% RSLogix 500 project I2P Project 01 - Tank 1 Process Control.RSS, saved by version 10.00.00.00 %
PROJECT "UNTITLED"    % processor: Bul.1763 MicroLogix 1100 Series B %

PROGRAM FILES
  LAD 2 "MAIN"  21 rungs  % Process Tank 1 Controls %
  LAD 3 "SIM"  18 rungs  % Simulation %

DATA FILES
  O0 OUTPUT  4 elements
  I1 INPUT  6 elements
  S2 STATUS  66 elements
  B3 BINARY  11 elements
  T4 TIMER  16 elements
  C5 COUNTER  1 elements
  R6 CONTROL  1 elements
  N7 INTEGER  1 elements
  F8 FLOAT  2 elements

LADDER 2 "MAIN"    % Process Tank 1 Controls %
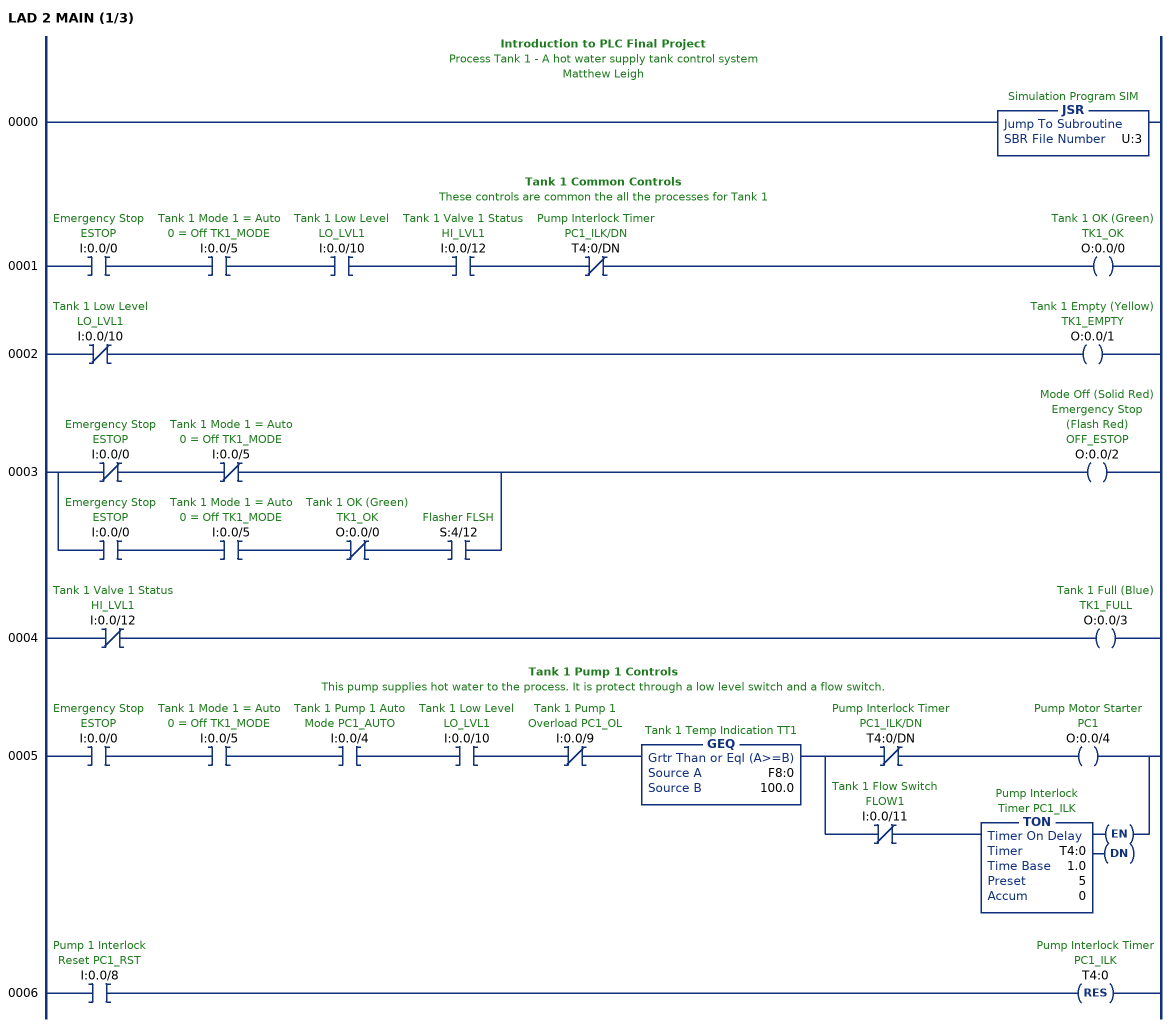
% Rung: 0 %
% TITLE: Introduction to PLC Final Project %
% Process Tank 1 - A hot water supply tank control system
% Matthew Leigh %
SOR JSR U:3 EOR
%   U:3  SIM  "Simulation Program" %
% Rung: 1 %
% TITLE: Tank 1 Common Controls %
% These controls are common the all the processes for Tank 1 %
SOR XIC I:0.0/0 XIC I:0.0/5 XIC I:0.0/10 XIC I:0.0/12 XIO T4:0/DN OTE O:0.0/0 EOR
%   I:0.0/0  ESTOP  "Emergency Stop" %
%   I:0.0/5  TK1_MODE  "Tank 1 Mode 1 = Auto 0 = Off" %
%   I:0.0/10  LO_LVL1  "Tank 1 Low Level" %
%   I:0.0/12  HI_LVL1  "Tank 1 Valve 1 Status" %
%   T4:0  PC1_ILK  "Pump Interlock Timer" %
%   O:0.0/0  TK1_OK  "Tank 1 OK (Green)" %
% Rung: 2 %
SOR XIO I:0.0/10 OTE O:0.0/1 EOR
%   I:0.0/10  LO_LVL1  "Tank 1 Low Level" %
%   O:0.0/1  TK1_EMPTY  "Tank 1 Empty (Yellow)" %
% Rung: 3 %
SOR BST XIO I:0.0/0 XIO I:0.0/5 NXB XIC I:0.0/0 XIC I:0.0/5 XIO O:0.0/0 XIC S:4/12 BND OTE O:0.0/2 EOR
%   I:0.0/0  ESTOP  "Emergency Stop" %
%   I:0.0/5  TK1_MODE  "Tank 1 Mode 1 = Auto 0 = Off" %
%   O:0.0/0  TK1_OK  "Tank 1 OK (Green)" %
%   S:4/12  FLSH  "Flasher" %
%   O:0.0/2  OFF_ESTOP  "Mode Off (Solid Red) Emergency Stop (Flash Red)" %
% Rung: 4 %
SOR XIO I:0.0/12 OTE O:0.0/3 EOR
%   I:0.0/12  HI_LVL1  "Tank 1 Valve 1 Status" %
%   O:0.0/3  TK1_FULL  "Tank 1 Full (Blue)" %
% Rung: 5 %
% TITLE: Tank 1 Pump 1 Controls %
% This pump supplies hot water to the process. It is protect through a low level switch and a flow switch. %
SOR XIC I:0.0/0 XIC I:0.0/5 XIC I:0.0/4 XIC I:0.0/10 XIO I:0.0/9 GEQ F8:0 100.0 BST XIO T4:0/DN OTE O:0.0/4 NXB XIO I:0.0/11 TON T4:0 1.0 5 0 BND EOR
%   I:0.0/0  ESTOP  "Emergency Stop" %
%   I:0.0/5  TK1_MODE  "Tank 1 Mode 1 = Auto 0 = Off" %
%   I:0.0/4  PC1_AUTO  "Tank 1 Pump 1 Auto Mode" %
%   I:0.0/10  LO_LVL1  "Tank 1 Low Level" %
%   I:0.0/9  PC1_OL  "Tank 1 Pump 1 Overload" %
%   F8:0  TT1  "Tank 1 Temp Indication" %
%   T4:0  PC1_ILK  "Pump Interlock Timer" %
%   O:0.0/4  PC1  "Pump Motor Starter" %
%   I:0.0/11  FLOW1  "Tank 1 Flow Switch" %
% Rung: 6 %
SOR XIC I:0.0/8 RES T4:0 EOR
%   I:0.0/8  PC1_RST  "Pump 1 Interlock Reset" %
%   T4:0  PC1_ILK  "Pump Interlock Timer" %

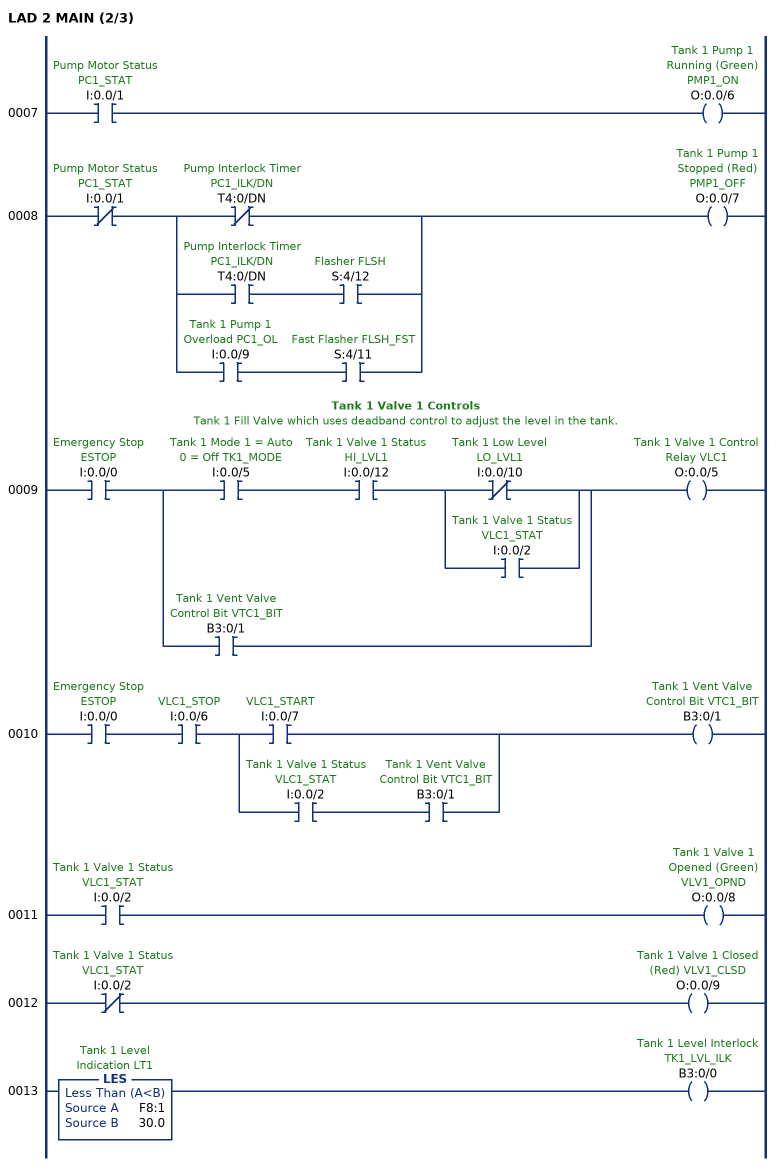
% Rung: 7 %
SOR XIC I:0.0/1 OTE O:0.0/6 EOR
%   I:0.0/1  PC1_STAT  "Pump Motor Status" %
%   O:0.0/6  PMP1_ON  "Tank 1 Pump 1 Running (Green)" %
% Rung: 8 %
SOR XIO I:0.0/1 BST XIO T4:0/DN NXB XIC T4:0/DN XIC S:4/12 NXB XIC I:0.0/9 XIC S:4/11 BND OTE O:0.0/7 EOR
%   I:0.0/1  PC1_STAT  "Pump Motor Status" %
%   T4:0  PC1_ILK  "Pump Interlock Timer" %
%   S:4/12  FLSH  "Flasher" %
%   I:0.0/9  PC1_OL  "Tank 1 Pump 1 Overload" %
%   S:4/11  FLSH_FST  "Fast Flasher" %
%   O:0.0/7  PMP1_OFF  "Tank 1 Pump 1 Stopped (Red)" %
% Rung: 9 %
% TITLE: Tank 1 Valve 1 Controls %
% Tank 1 Fill Valve which uses deadband control to adjust the level in the tank. %
SOR XIC I:0.0/0 BST XIC I:0.0/5 XIC I:0.0/12 BST XIO I:0.0/10 NXB XIC I:0.0/2 BND NXB XIC B3:0/1 BND OTE O:0.0/5 EOR
%   I:0.0/0  ESTOP  "Emergency Stop" %
%   I:0.0/5  TK1_MODE  "Tank 1 Mode 1 = Auto 0 = Off" %
%   I:0.0/12  HI_LVL1  "Tank 1 Valve 1 Status" %
%   I:0.0/10  LO_LVL1  "Tank 1 Low Level" %
%   I:0.0/2  VLC1_STAT  "Tank 1 Valve 1 Status" %
%   B3:0/1  VTC1_BIT  "Tank 1 Vent Valve Control Bit" %
%   O:0.0/5  VLC1  "Tank 1 Valve 1 Control Relay" %
% Rung: 10 %
SOR XIC I:0.0/0 XIC I:0.0/6 BST XIC I:0.0/7 NXB XIC I:0.0/2 XIC B3:0/1 BND OTE B3:0/1 EOR
%   I:0.0/0  ESTOP  "Emergency Stop" %
%   I:0.0/6  VLC1_STOP %
%   I:0.0/7  VLC1_START %
%   I:0.0/2  VLC1_STAT  "Tank 1 Valve 1 Status" %
%   B3:0/1  VTC1_BIT  "Tank 1 Vent Valve Control Bit" %
% Rung: 11 %
SOR XIC I:0.0/2 OTE O:0.0/8 EOR
%   I:0.0/2  VLC1_STAT  "Tank 1 Valve 1 Status" %
%   O:0.0/8  VLV1_OPND  "Tank 1 Valve 1 Opened (Green)" %
% Rung: 12 %
SOR XIO I:0.0/2 OTE O:0.0/9 EOR
%   I:0.0/2  VLC1_STAT  "Tank 1 Valve 1 Status" %
%   O:0.0/9  VLV1_CLSD  "Tank 1 Valve 1 Closed (Red)" %
% Rung: 13 %
SOR LES F8:1 30.0 OTE B3:0/0 EOR
%   F8:1  LT1  "Tank 1 Level Indication" %
%   B3:0/0  TK1_LVL_ILK  "Tank 1 Level Interlock" %

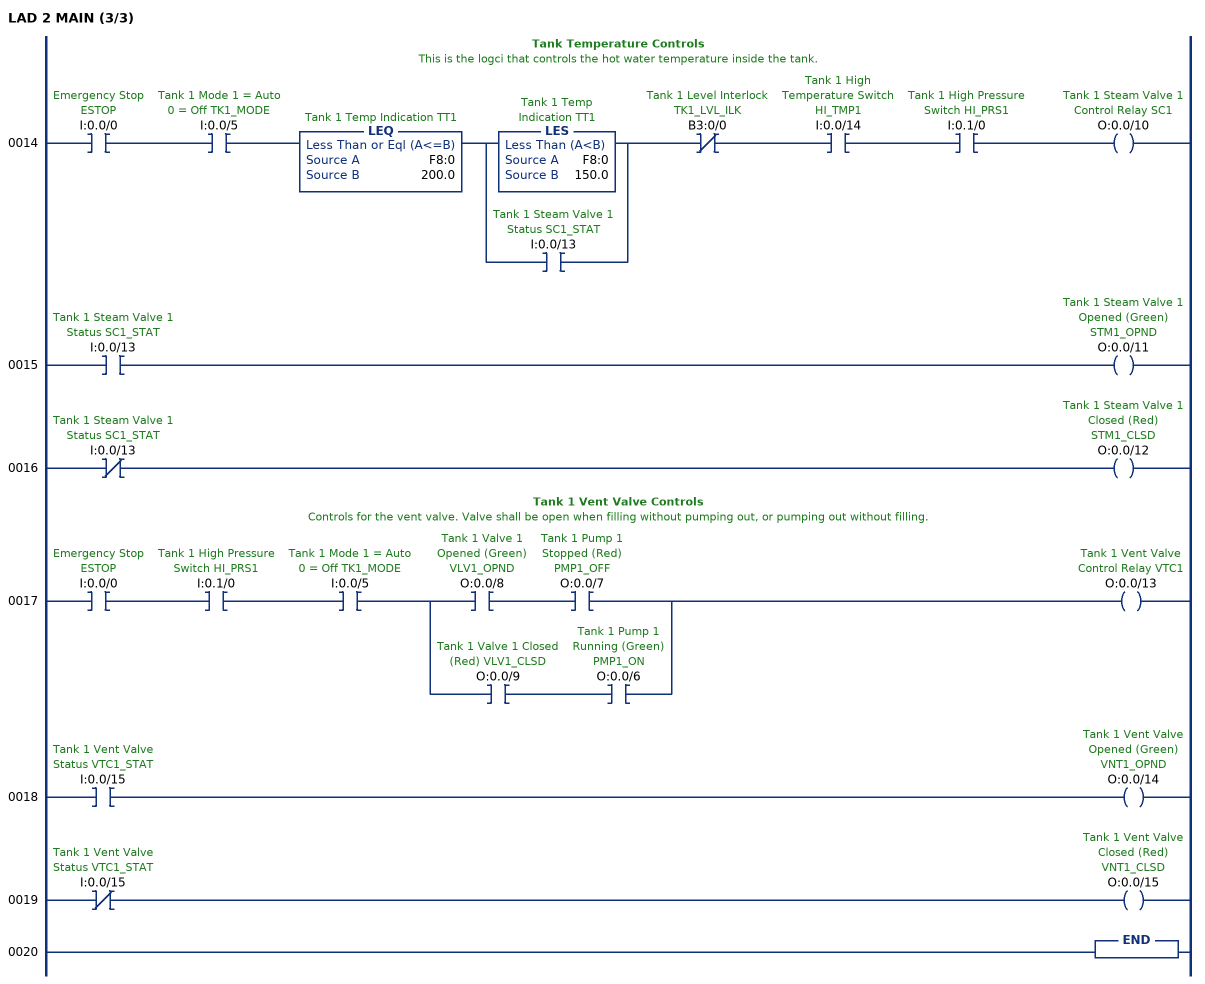
% Rung: 14 %
% TITLE: Tank Temperature Controls %
% This is the logci that controls the hot water temperature inside the tank. %
SOR XIC I:0.0/0 XIC I:0.0/5 LEQ F8:0 200.0 BST LES F8:0 150.0 NXB XIC I:0.0/13 BND XIO B3:0/0 XIC I:0.0/14 XIC I:0.1/0 OTE O:0.0/10 EOR
%   I:0.0/0  ESTOP  "Emergency Stop" %
%   I:0.0/5  TK1_MODE  "Tank 1 Mode 1 = Auto 0 = Off" %
%   F8:0  TT1  "Tank 1 Temp Indication" %
%   I:0.0/13  SC1_STAT  "Tank 1 Steam Valve 1 Status" %
%   B3:0/0  TK1_LVL_ILK  "Tank 1 Level Interlock" %
%   I:0.0/14  HI_TMP1  "Tank 1 High Temperature Switch" %
%   I:0.1/0  HI_PRS1  "Tank 1 High Pressure Switch" %
%   O:0.0/10  SC1  "Tank 1 Steam Valve 1 Control Relay" %
% Rung: 15 %
SOR XIC I:0.0/13 OTE O:0.0/11 EOR
%   I:0.0/13  SC1_STAT  "Tank 1 Steam Valve 1 Status" %
%   O:0.0/11  STM1_OPND  "Tank 1 Steam Valve 1 Opened (Green)" %
% Rung: 16 %
SOR XIO I:0.0/13 OTE O:0.0/12 EOR
%   I:0.0/13  SC1_STAT  "Tank 1 Steam Valve 1 Status" %
%   O:0.0/12  STM1_CLSD  "Tank 1 Steam Valve 1 Closed (Red)" %
% Rung: 17 %
% TITLE: Tank 1 Vent Valve Controls %
% Controls for the vent valve. Valve shall be open when filling without pumping out, or pumping out without filling. %
SOR XIC I:0.0/0 XIC I:0.1/0 XIC I:0.0/5 BST XIC O:0.0/8 XIC O:0.0/7 NXB XIC O:0.0/9 XIC O:0.0/6 BND OTE O:0.0/13 EOR
%   I:0.0/0  ESTOP  "Emergency Stop" %
%   I:0.1/0  HI_PRS1  "Tank 1 High Pressure Switch" %
%   I:0.0/5  TK1_MODE  "Tank 1 Mode 1 = Auto 0 = Off" %
%   O:0.0/8  VLV1_OPND  "Tank 1 Valve 1 Opened (Green)" %
%   O:0.0/7  PMP1_OFF  "Tank 1 Pump 1 Stopped (Red)" %
%   O:0.0/9  VLV1_CLSD  "Tank 1 Valve 1 Closed (Red)" %
%   O:0.0/6  PMP1_ON  "Tank 1 Pump 1 Running (Green)" %
%   O:0.0/13  VTC1  "Tank 1 Vent Valve Control Relay" %
% Rung: 18 %
SOR XIC I:0.0/15 OTE O:0.0/14 EOR
%   I:0.0/15  VTC1_STAT  "Tank 1 Vent Valve Status" %
%   O:0.0/14  VNT1_OPND  "Tank 1 Vent Valve Opened (Green)" %
% Rung: 19 %
SOR XIO I:0.0/15 OTE O:0.0/15 EOR
%   I:0.0/15  VTC1_STAT  "Tank 1 Vent Valve Status" %
%   O:0.0/15  VNT1_CLSD  "Tank 1 Vent Valve Closed (Red)" %
% Rung: 20 %
SOR END EOR

LADDER 3 "SIM"    % Simulation %
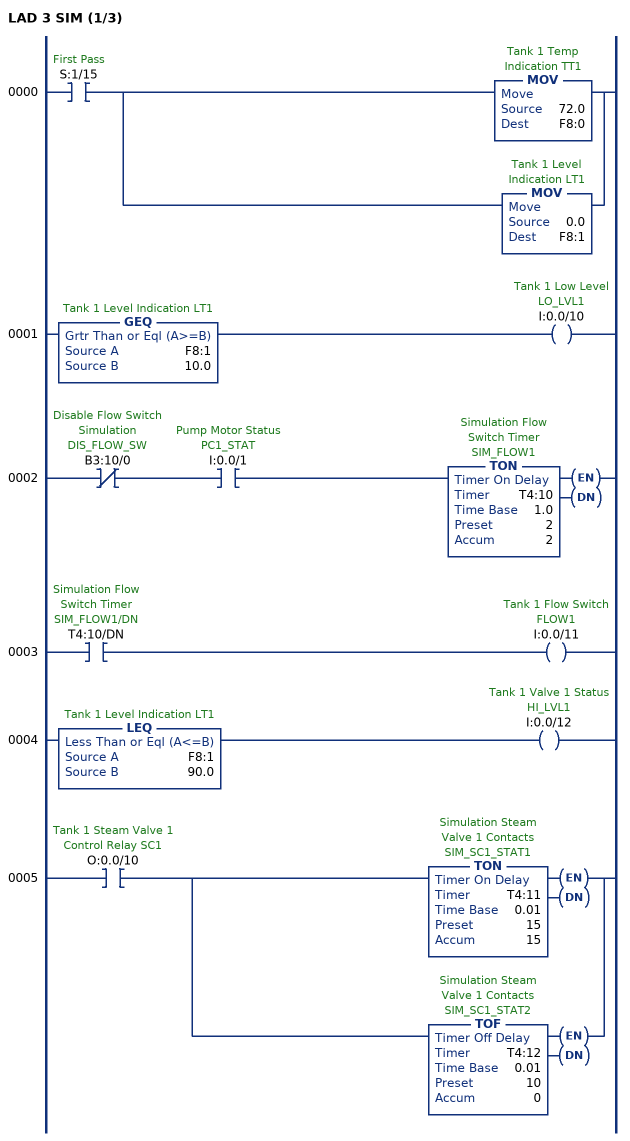
% Rung: 0 %
SOR XIC S:1/15 BST MOV 72.0 F8:0 NXB MOV 0.0 F8:1 BND EOR
%   S:1/15  "First Pass" %
%   F8:0  TT1  "Tank 1 Temp Indication" %
%   F8:1  LT1  "Tank 1 Level Indication" %
% Rung: 1 %
SOR GEQ F8:1 10.0 OTE I:0.0/10 EOR
%   F8:1  LT1  "Tank 1 Level Indication" %
%   I:0.0/10  LO_LVL1  "Tank 1 Low Level" %
% Rung: 2 %
SOR XIO B3:10/0 XIC I:0.0/1 TON T4:10 1.0 2 2 EOR
%   B3:10/0  DIS_FLOW_SW  "Disable Flow Switch Simulation" %
%   I:0.0/1  PC1_STAT  "Pump Motor Status" %
%   T4:10  SIM_FLOW1  "Simulation Flow Switch Timer" %
% Rung: 3 %
SOR XIC T4:10/DN OTE I:0.0/11 EOR
%   T4:10  SIM_FLOW1  "Simulation Flow Switch Timer" %
%   I:0.0/11  FLOW1  "Tank 1 Flow Switch" %
% Rung: 4 %
SOR LEQ F8:1 90.0 OTE I:0.0/12 EOR
%   F8:1  LT1  "Tank 1 Level Indication" %
%   I:0.0/12  HI_LVL1  "Tank 1 Valve 1 Status" %
% Rung: 5 %
SOR XIC O:0.0/10 BST TON T4:11 0.01 15 15 NXB TOF T4:12 0.01 10 0 BND EOR
%   O:0.0/10  SC1  "Tank 1 Steam Valve 1 Control Relay" %
%   T4:11  SIM_SC1_STAT1  "Simulation Steam Valve 1 Contacts" %
%   T4:12  SIM_SC1_STAT2  "Simulation Steam Valve 1 Contacts" %

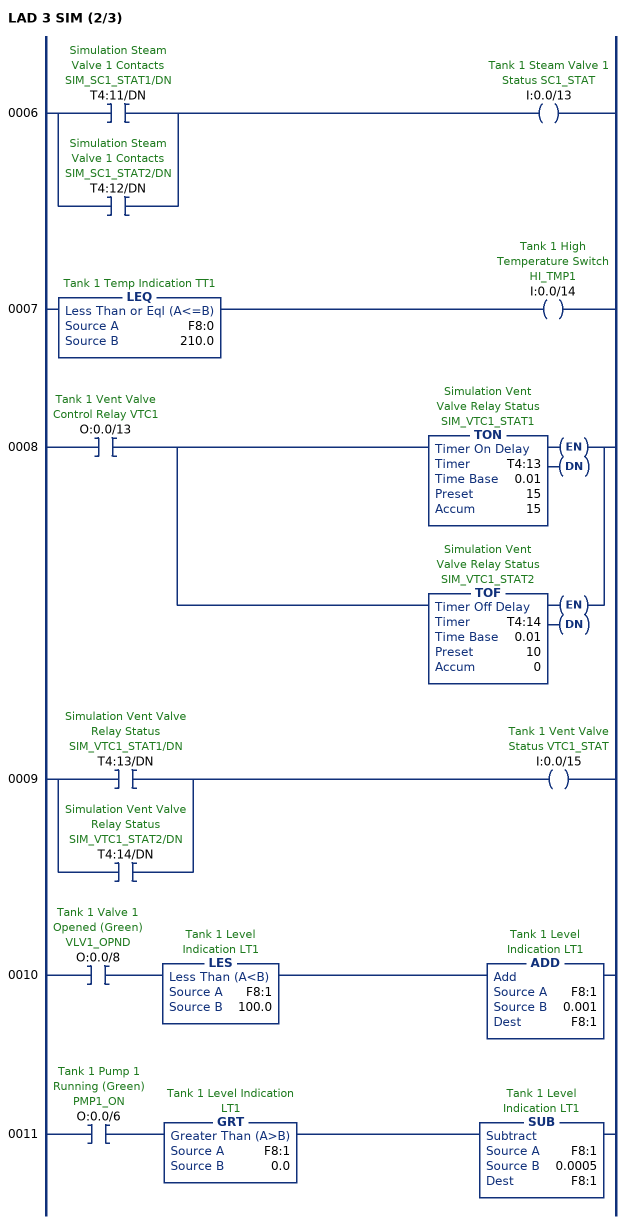
% Rung: 6 %
SOR BST XIC T4:11/DN NXB XIC T4:12/DN BND OTE I:0.0/13 EOR
%   T4:11  SIM_SC1_STAT1  "Simulation Steam Valve 1 Contacts" %
%   T4:12  SIM_SC1_STAT2  "Simulation Steam Valve 1 Contacts" %
%   I:0.0/13  SC1_STAT  "Tank 1 Steam Valve 1 Status" %
% Rung: 7 %
SOR LEQ F8:0 210.0 OTE I:0.0/14 EOR
%   F8:0  TT1  "Tank 1 Temp Indication" %
%   I:0.0/14  HI_TMP1  "Tank 1 High Temperature Switch" %
% Rung: 8 %
SOR XIC O:0.0/13 BST TON T4:13 0.01 15 15 NXB TOF T4:14 0.01 10 0 BND EOR
%   O:0.0/13  VTC1  "Tank 1 Vent Valve Control Relay" %
%   T4:13  SIM_VTC1_STAT1  "Simulation Vent Valve Relay Status" %
%   T4:14  SIM_VTC1_STAT2  "Simulation Vent Valve Relay Status" %
% Rung: 9 %
SOR BST XIC T4:13/DN NXB XIC T4:14/DN BND OTE I:0.0/15 EOR
%   T4:13  SIM_VTC1_STAT1  "Simulation Vent Valve Relay Status" %
%   T4:14  SIM_VTC1_STAT2  "Simulation Vent Valve Relay Status" %
%   I:0.0/15  VTC1_STAT  "Tank 1 Vent Valve Status" %
% Rung: 10 %
SOR XIC O:0.0/8 LES F8:1 100.0 ADD F8:1 0.001 F8:1 EOR
%   O:0.0/8  VLV1_OPND  "Tank 1 Valve 1 Opened (Green)" %
%   F8:1  LT1  "Tank 1 Level Indication" %
% Rung: 11 %
SOR XIC O:0.0/6 GRT F8:1 0.0 SUB F8:1 0.0005 F8:1 EOR
%   O:0.0/6  PMP1_ON  "Tank 1 Pump 1 Running (Green)" %
%   F8:1  LT1  "Tank 1 Level Indication" %

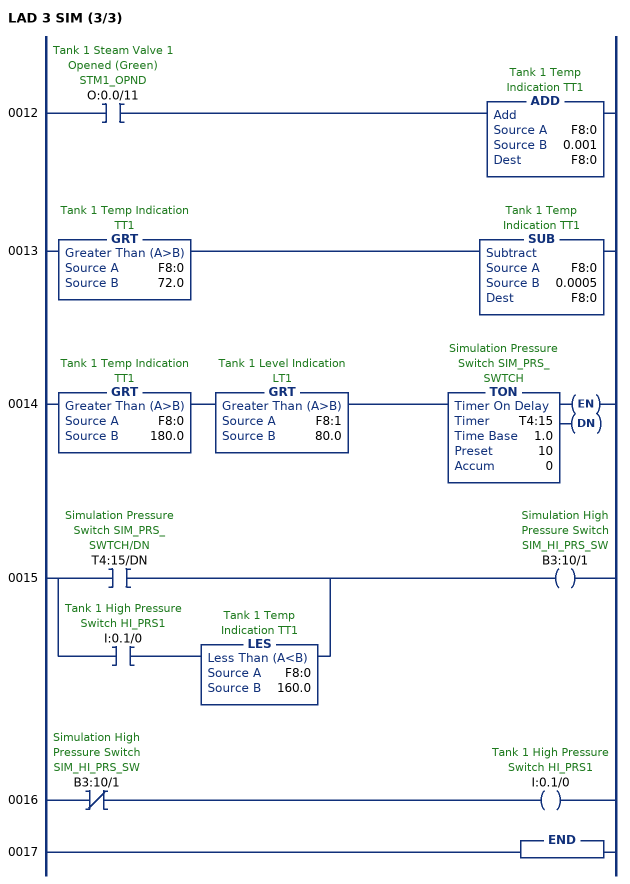
% Rung: 12 %
SOR XIC O:0.0/11 ADD F8:0 0.001 F8:0 EOR
%   O:0.0/11  STM1_OPND  "Tank 1 Steam Valve 1 Opened (Green)" %
%   F8:0  TT1  "Tank 1 Temp Indication" %
% Rung: 13 %
SOR GRT F8:0 72.0 SUB F8:0 0.0005 F8:0 EOR
%   F8:0  TT1  "Tank 1 Temp Indication" %
% Rung: 14 %
SOR GRT F8:0 180.0 GRT F8:1 80.0 TON T4:15 1.0 10 0 EOR
%   F8:0  TT1  "Tank 1 Temp Indication" %
%   F8:1  LT1  "Tank 1 Level Indication" %
%   T4:15  SIM_PRS_SWTCH  "Simulation Pressure Switch" %
% Rung: 15 %
SOR BST XIC T4:15/DN NXB XIC I:0.1/0 LES F8:0 160.0 BND OTE B3:10/1 EOR
%   T4:15  SIM_PRS_SWTCH  "Simulation Pressure Switch" %
%   I:0.1/0  HI_PRS1  "Tank 1 High Pressure Switch" %
%   F8:0  TT1  "Tank 1 Temp Indication" %
%   B3:10/1  SIM_HI_PRS_SW  "Simulation High Pressure Switch" %
% Rung: 16 %
SOR XIO B3:10/1 OTE I:0.1/0 EOR
%   B3:10/1  SIM_HI_PRS_SW  "Simulation High Pressure Switch" %
%   I:0.1/0  HI_PRS1  "Tank 1 High Pressure Switch" %
% Rung: 17 %
SOR END EOR

OTHER DOCUMENTED ADDRESSES
  I:0.0/3  PC1_HAND  "Tank 1 Pump 1 Mode Hand"
  S:4/13  FLSH_SLO  "Slow Flasher"

DATA TABLE (non-zero values as saved)
DATA T4
% .PRE .ACC %
% T4:0 % 5 0
% T4:10 % 2 2
% T4:11 % 15 15
% T4:12 % 10 0
% T4:13 % 15 15
% T4:14 % 10 0
% T4:15 % 10 0
DATA F8
% F8:0 % 154.2602 75.46014
